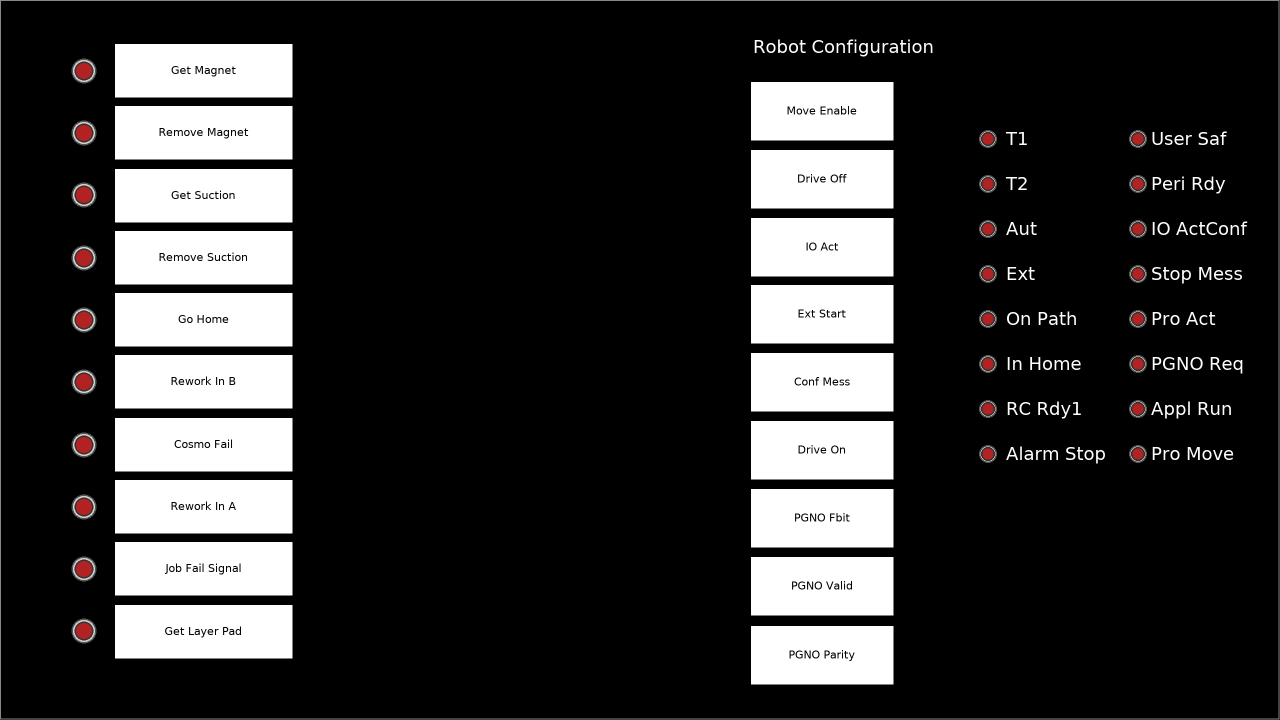
VISUALIZATION PAGE_KR1  // 1280x720
    Lamp1 (64,57 40x28), variable: KR1.bInBit[3,0], style: Lamp-Lamp1-Red
    Lamp1 (64,119 40x28), variable: KR1.bInBit[3,1], style: Lamp-Lamp1-Red
    Lamp1 (64,181 40x28), variable: KR1.bInBit[3,2], style: Lamp-Lamp1-Red
    Lamp1 (64,244 40x28), variable: KR1.bInBit[3,3], style: Lamp-Lamp1-Red
    Lamp1 (64,306 40x28), variable: KR1.bInBit[3,4], style: Lamp-Lamp1-Red
    Lamp1 (64,368 40x28), variable: KR1.bInBit[3,5], style: Lamp-Lamp1-Red
    Lamp1 (64,431 40x28), variable: KR1.bInBit[3,6], style: Lamp-Lamp1-Red
    Lamp1 (64,493 40x28), variable: KR1.bInBit[3,7], style: Lamp-Lamp1-Red
    RoundedRectangle (114,43 179x55), "Get Magnet"
        toggle KR1.bOutBit[3,0]
        OnMouseClick: execute { GVL.KR1_EOAT_FILL := true; }
    RoundedRectangle (114,105 179x55), "Remove Magnet"
        toggle KR1.bOutBit[3,1]
        OnMouseClick: execute { GVL.KR1_EOAT_FILL := false; }
    RoundedRectangle (114,168 179x55), "Get Suction"
        toggle KR1.bOutBit[3,2]
        OnMouseClick: execute { GVL.KR1_EOAT_SUCTION := true; }
    RoundedRectangle (114,230 179x55), "Remove Suction"
        toggle KR1.bOutBit[3,3]
        OnMouseClick: execute { GVL.KR1_EOAT_SUCTION := false; }
    RoundedRectangle (114,292 179x55), "Go Home"
        toggle KR1.bOutBit[3,4]
        OnMouseClick: execute {  }
    RoundedRectangle (114,354 179x55), "Rework In B"
        toggle KR1.bOutBit[3,5]
        OnMouseClick: execute {  }
    RoundedRectangle (114,417 179x55), "Cosmo Fail"
        toggle KR1.bOutBit[3,6]
        OnMouseClick: execute {  }
    RoundedRectangle (114,479 179x55), "Rework In A"
        toggle KR1.bOutBit[3,7]
        OnMouseClick: execute {  }
    RoundedRectangle (114,541 179x55), "Job Fail Signal"
        toggle KR1.bOutBit[4,0]
        OnMouseClick: execute {  }
    RoundedRectangle (114,604 179x55), "Get Layer Pad"
        toggle KR1.bOutBit[4,1]
        OnMouseClick: execute {  }
    Lamp1 (64,555 40x28), variable: KR1.bInBit[4,0], style: Lamp-Lamp1-Red
    Lamp1 (64,617 40x28), variable: KR1.bInBit[4,1], style: Lamp-Lamp1-Red
    RoundedRectangle (750,81 144x60), "Move Enable"
        toggle KR1.bOutBit[1,0]
        OnMouseClick: execute {  }
    RoundedRectangle (750,149 144x60), "Drive Off"
        toggle KR1.bOutBit[1,1]
        OnMouseClick: execute {  }
    RoundedRectangle (750,217 144x60), "IO Act"
        toggle KR1.bOutBit[1,2]
        OnMouseClick: execute {  }
    RoundedRectangle (750,284 144x60), "Ext Start"
        toggle KR1.bOutBit[1,3]
        OnMouseClick: execute {  }
    RoundedRectangle (750,352 144x60), "Conf Mess"
        toggle KR1.bOutBit[1,4]
        OnMouseClick: execute {  }
    RoundedRectangle (750,420 144x60), "Drive On"
        toggle KR1.bOutBit[1,5]
        OnMouseClick: execute {  }
    RoundedRectangle (750,488 144x60), "PGNO Fbit"
        toggle KR1.bOutBit[1,6]
        OnMouseClick: execute {  }
    RoundedRectangle (750,556 144x60), "PGNO Valid"
        toggle KR1.bOutBit[1,7]
        OnMouseClick: execute {  }
    RoundedRectangle (750,625 144x60), "PGNO Parity"
        toggle KR1.bOutBit[2,0]
        OnMouseClick: execute {  }
    Lamp1 (978,129 20x20), variable: KR1.bInBit[1,0], style: Lamp-Lamp1-Red
    Lamp1 (978,174 20x20), variable: KR1.bInBit[1,1], style: Lamp-Lamp1-Red
    Lamp1 (978,219 20x20), variable: KR1.bInBit[1,2], style: Lamp-Lamp1-Red
    Lamp1 (978,264 20x20), variable: KR1.bInBit[1,3], style: Lamp-Lamp1-Red
    Lamp1 (978,309 20x20), variable: KR1.bInBit[1,4], style: Lamp-Lamp1-Red
    Lamp1 (978,354 20x20), variable: KR1.bInBit[1,5], style: Lamp-Lamp1-Red
    Lamp1 (978,399 20x20), variable: KR1.bInBit[1,6], style: Lamp-Lamp1-Red
    Lamp1 (978,444 20x20), variable: KR1.bInBit[1,7], style: Lamp-Lamp1-Red
    Label (1003,124 105x30), "T1"
    Label (1003,169 105x30), "T2"
    Label (1003,214 105x30), "Aut"
    Label (1003,259 105x30), "Ext"
    Label (1003,304 105x30), "On Path"
    Label (1003,349 105x30), "In Home"
    Label (1003,394 105x30), "RC Rdy1"
    Label (1003,439 105x30), "Alarm Stop"
    Lamp1 (1128,129 20x20), variable: KR1.bInBit[2,0], style: Lamp-Lamp1-Red
    Lamp1 (1128,174 20x20), variable: KR1.bInBit[2,1], style: Lamp-Lamp1-Red
    Lamp1 (1128,219 20x20), variable: KR1.bInBit[2,2], style: Lamp-Lamp1-Red
    Lamp1 (1128,264 20x20), variable: KR1.bInBit[2,3], style: Lamp-Lamp1-Red
    Lamp1 (1128,309 20x20), variable: KR1.bInBit[2,4], style: Lamp-Lamp1-Red
    Lamp1 (1128,354 20x20), variable: KR1.bInBit[2,5], style: Lamp-Lamp1-Red
    Lamp1 (1128,399 20x20), variable: KR1.bInBit[2,6], style: Lamp-Lamp1-Red
    Lamp1 (1128,444 20x20), variable: KR1.bInBit[2,7], style: Lamp-Lamp1-Red
    Label (1148,124 110x30), "User Saf"
    Label (1148,169 110x30), "Peri Rdy"
    Label (1148,214 110x30), "IO ActConf"
    Label (1148,259 110x30), "Stop Mess"
    Label (1148,304 110x30), "Pro Act"
    Label (1148,349 110x30), "PGNO Req"
    Label (1148,394 110x30), "Appl Run"
    Label (1148,439 110x30), "Pro Move"
    Label (750,32 250x30), "Robot Configuration"
END_VISUALIZATION

(* stored: Version 1.1.0.1, ProductVersion 3.1.4024.12
   Visu PAGE_KR1: Id {8b90c252-6767-4a57-a246-d2639796ea7f} *)
